INTERFACE I_AnalogDevice

PROPERTY ModuleType : REFERENCE TO STRING
GET
END_GET
END_PROPERTY

METHOD MR_FirstCycle : BOOL
VAR_INPUT
	sName 			: STRING;
	sModuleType 	: STRING;
	sPortID			: STRING;
END_VAR
END_METHOD

PROPERTY Name : REFERENCE TO STRING
GET
END_GET
END_PROPERTY

PROPERTY PortID : REFERENCE TO STRING
GET
END_GET
END_PROPERTY

END_INTERFACE

(* stored: Version 1.1.0.1, ProductVersion 3.1.4024.9
   Itf I_AnalogDevice: Id {bcdc6111-eaee-4f4e-8af8-6ec1fa8517af}
   Property ModuleType: Id {c25d43fb-c611-4c24-92f2-1eceb69e3664}
   Get Get: Id {6ce7e59e-fb9b-4b66-a61a-80e005060733}
   Method MR_FirstCycle: Id {8332a5e3-e038-4fad-b817-d3606ea1dff7}
   Property Name: Id {967fb438-0f17-4cb8-9fc5-cebf3a5ac313}
   Get Get: Id {d5551de7-307e-4c8f-8951-6650a1cbbee2}
   Property PortID: Id {e3568c8b-ba97-4f60-9a28-58b8894dbf75}
   Get Get: Id {0bae3160-5073-4402-bbe5-5eb070fea5f1} *)
